// TIA Portal V20 export
TYPE "typeSequenceControlNodeJobInterface_sideTapeAttachment"
// stored: Namespace Unit1.Em4
   STRUCT
      rightTapeGetJob2 : "LER_typeJobInterface";
      leftTapeGetJob3 : "LER_typeJobInterface";
      tape1PutJob4 : "LER_typeJobInterface";
      tape2PutJob5 : "LER_typeJobInterface";
      tape3PutJob6 : "LER_typeJobInterface";
      tape4PutJob7 : "LER_typeJobInterface";
      TapeIdleJob8 { S7_SetPoint := 'True'} : "LER_typeJobInterface";
   END_STRUCT;
END_TYPE
